FUNCTION_BLOCK BoxDropper_SIFB
  (* Standard: 61499-2 *)
  (* Version 0.1, 2016-00-08, hpea485, UOA *)
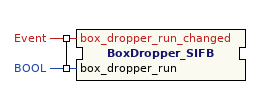
  EVENT_INPUT
    box_dropper_run_changed WITH box_dropper_run;
  END_EVENT
  VAR_INPUT
    box_dropper_run : BOOL;
  END_VAR
  VAR
    tx_box_dropper_run : BOOL; (* TOPIO_OUT *)
  END_VAR
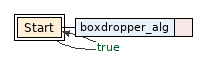
  EC_STATES
    Start : boxdropper_alg;
  END_STATES
  EC_TRANSITIONS
    Start TO Start := true;
  END_TRANSITIONS
  ALGORITHM boxdropper_alg IN VHDL:
tx_box_dropper <= box_dropper;
DONE <= '1';
  END_ALGORITHM
END_FUNCTION_BLOCK
